Yaskawa INFORM job: SBTCLOSE.JBI

/JOB
//NAME SBTCLOSE
//POS
///NPOS 0,0,0,0,0,0
//INST
///DATE 2020/09/25 15:30
///ATTR SC,RW,MC
///GROUP1 RB1
///LVARS 0,0,1,0,1,0,0,0
NOP
SET B069 0
SKILLSND "SpeedbotClose"
end
